Fanuc KAREL source: kb00178.KL

-- PROVISIONAL review KL for V1013-1; original PC SHA256 a85e8f0b8c70f1f68ff1f9577b4a9a529eab082441b39cd16e8738b6a9d803b1
-- Incomplete behavior may be omitted. Consult companion uncertainty JSON. Do not deploy.
PROGRAM KB00178
%NOLOCKGROUP
BEGIN
  -- UNRESOLVED_PC offsets 5-12; opcodes 9D,23
  -- UNRESOLVED_PC offsets 17-28; opcodes 2E,23
  -- UNRESOLVED_PC offsets 33-40; opcodes 9D,23
  -- UNRESOLVED_PC offsets 45-67; opcodes 27,22,22,22,31
  -- UNRESOLVED_PC offsets 72-76; opcodes 7F
END KB00178
